{attribute addProperty BoxType "ATH2000-0250-0022"}
{attribute addProperty Id "A_0014_ATH2050_5501_0022ATH2050_3A2EE8A79812.25"}
{attribute addProperty CRC "539192398"}
{attribute addProperty SizeInBites "98"}
{attribute addProperty SizeInBytes "12.25"}
TYPE A_0001_ATH2000_0250_0022_20236C4E EXTENDS ATH2000_BA5A9548 :
STRUCT
	{attribute addProperty Name "A_0014_ATH2050_5501_0022"}
	A_0014_ATH2050_5501_0022 : ATH2050_3A2EE8A7;
END_STRUCT
END_TYPE

(* stored: Version 1.2.0.0, ProductVersion 3.1.4024.9
   DUT A_0001_ATH2000_0250_0022_20236C4E: Id {ab44b827-53fe-4075-907b-b121c1824839} *)
